ABB RAPID module: RotationTopDownTraj.MOD

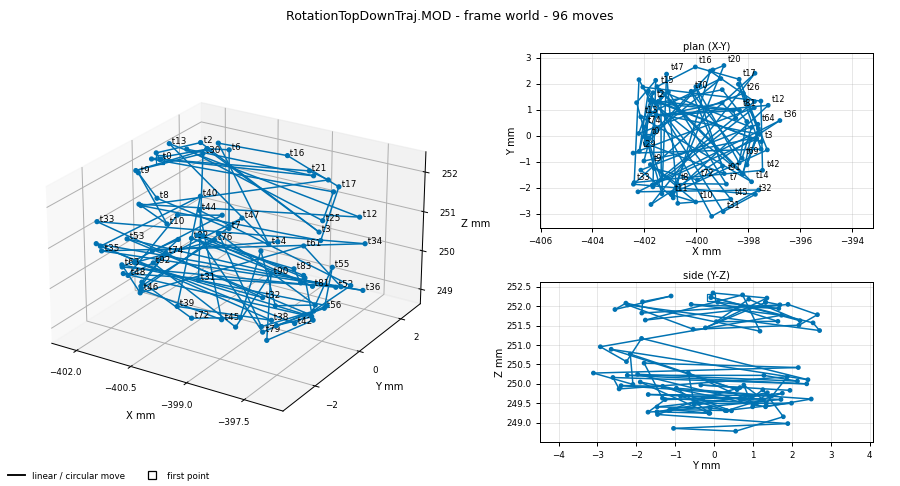
[picture p0: tool path of RotationTopDownTraj.MOD in frame world, 96 of 97 moves have a stored position in this frame; points joined in program order, loops and branches not executed]
MODULE MainModule
PERS tooldata Servo:=[TRUE,[[0,0,114.2],[1,0,0,0]],[0.215,[8.7,12.3,49.2],[1,0,0,0],0.00021,0.00024,0.00009]];
PERS tooldata tObject:=[TRUE,[[0,0,130],[0.707106781,-0.707106781,0,0]],[0.215,[8.7,12.3,49.2],[1,0,0,0],0.00021,0.00024,0.00009]];
PERS wobjdata handpos:= [FALSE,TRUE,"",[[-400,0,250],[1,0,0,0]],[[0,0,0],[1,0,0,0]]];
    PROC main()
        ConfL\Off;
        SingArea\Wrist;
        !Startpos
        MoveAbsJ [[0.441359,-16.418,10.8814,2.79121,60.2034,-14.3875],[168.362,9E+09,9E+09,9E+09,9E+09,9E+09]] \NoEOffs, v1000, fine, wi_tGripper;
        path;
    ENDPROC
    PROC path()

VAR robtarget t0 := [[-1.8594772767669543, -0.08634270627151014, 2.220359244544771], [1,0,0,0], [0,0,-1,4], [-96,9E+09,9E+09,9E+09,9E+09,9E+09]];
VAR robtarget t1 := [[-1.9968136850268585, -0.031200990620815494, 2.337895466549644], [1,0,0,0], [0,0,-1,4], [-96,9E+09,9E+09,9E+09,9E+09,9E+09]];
VAR robtarget t2 := [[-1.664406335824331, 1.3530457056262837, 2.2071876558339123], [1,0,0,0], [0,0,-1,4], [-96,9E+09,9E+09,9E+09,9E+09,9E+09]];
VAR robtarget t3 := [[2.5103465951354025, -0.22605266531133467, 1.4426248167740197], [1,0,0,0], [0,0,-1,4], [-96,9E+09,9E+09,9E+09,9E+09,9E+09]];
VAR robtarget t4 := [[-1.4698118716392545, 1.3182294867649416, 2.0926888140146214], [1,0,0,0], [0,0,-1,4], [-96,9E+09,9E+09,9E+09,9E+09,9E+09]];
VAR robtarget t5 := [[-1.4558740515764113, 1.316986954334625, 2.106495340552807], [1,0,0,0], [0,0,-1,4], [-96,9E+09,9E+09,9E+09,9E+09,9E+09]];
VAR robtarget t6 := [[-1.0750677254328767, 1.687805937624978, 2.033368826106924], [1,0,0,0], [0,0,-1,4], [-96,9E+09,9E+09,9E+09,9E+09,9E+09]];
VAR robtarget t7 := [[1.1584643511839996, -1.860619126747291, 1.8215288250970674], [1,0,0,0], [0,0,-1,4], [-96,9E+09,9E+09,9E+09,9E+09,9E+09]];
VAR robtarget t8 := [[-0.7602163155200519, -1.8412191017858337, 2.1115963079865545], [1,0,0,0], [0,0,-1,4], [-96,9E+09,9E+09,9E+09,9E+09,9E+09]];
VAR robtarget t9 := [[-1.767026063291215, -1.108222633044502, 2.2588988392369096], [1,0,0,0], [0,0,-1,4], [-96,9E+09,9E+09,9E+09,9E+09,9E+09]];
VAR robtarget t10 := [[-0.021667862335108423, -2.550518737223798, 1.91242402643374], [1,0,0,0], [0,0,-1,4], [-96,9E+09,9E+09,9E+09,9E+09,9E+09]];
VAR robtarget t11 := [[-0.9577512947057534, -2.269361244202862, 2.075411818055441], [1,0,0,0], [0,0,-1,4], [-96,9E+09,9E+09,9E+09,9E+09,9E+09]];
VAR robtarget t12 := [[2.769781059373928, 1.1748233186231039, 1.355829415691719], [1,0,0,0], [0,0,-1,4], [-96,9E+09,9E+09,9E+09,9E+09,9E+09]];
VAR robtarget t13 := [[-2.139028394244537, 0.7292214301304468, 2.2879263104279], [1,0,0,0], [0,0,-1,4], [-96,9E+09,9E+09,9E+09,9E+09,9E+09]];
VAR robtarget t14 := [[2.1287073060742876, -1.7703456012939633, 1.6407871642460183], [1,0,0,0], [0,0,-1,4], [-96,9E+09,9E+09,9E+09,9E+09,9E+09]];
VAR robtarget t15 := [[-1.513174804260462, 1.8955196047121665, 2.0442006001312616], [1,0,0,0], [0,0,-1,4], [-96,9E+09,9E+09,9E+09,9E+09,9E+09]];
VAR robtarget t16 := [[-0.03680877924259918, 2.6515244667226368, 1.7794670852935306], [1,0,0,0], [0,0,-1,4], [-96,9E+09,9E+09,9E+09,9E+09,9E+09]];
VAR robtarget t17 := [[1.6507116212087651, 2.1766451428121156, 1.5087291037843746], [1,0,0,0], [0,0,-1,4], [-96,9E+09,9E+09,9E+09,9E+09,9E+09]];
VAR robtarget t18 := [[2.735569481461933, -0.5419181356070709, 1.40601519419272], [1,0,0,0], [0,0,-1,4], [-96,9E+09,9E+09,9E+09,9E+09,9E+09]];
VAR robtarget t19 := [[-0.9380260342751103, -2.219623851546317, 2.029077273537317], [1,0,0,0], [0,0,-1,4], [-96,9E+09,9E+09,9E+09,9E+09,9E+09]];
VAR robtarget t20 := [[1.0643405616793875, 2.7065514744939527, 1.3718604556537926], [1,0,0,0], [0,0,-1,4], [-96,9E+09,9E+09,9E+09,9E+09,9E+09]];
VAR robtarget t21 := [[0.6390066698048532, 2.5391954277440463, 1.5687647182886193], [1,0,0,0], [0,0,-1,4], [-96,9E+09,9E+09,9E+09,9E+09,9E+09]];
VAR robtarget t22 := [[-1.8474595325347547, -0.0769827159651687, 2.225891768617379], [1,0,0,0], [0,0,-1,4], [-96,9E+09,9E+09,9E+09,9E+09,9E+09]];
VAR robtarget t23 := [[0.9480233018981318, 2.2051691359949985, 1.6252779556548258], [1,0,0,0], [0,0,-1,4], [-96,9E+09,9E+09,9E+09,9E+09,9E+09]];
VAR robtarget t24 := [[-1.7519363441106846, 0.8872878448625607, 2.1765162636907256], [1,0,0,0], [0,0,-1,4], [-96,9E+09,9E+09,9E+09,9E+09,9E+09]];
VAR robtarget t25 := [[2.439463854161823, 0.05449093458225296, 1.6002323474520679], [1,0,0,0], [0,0,-1,4], [-96,9E+09,9E+09,9E+09,9E+09,9E+09]];
VAR robtarget t26 := [[1.8136195796860872, 1.635838943826832, 1.607891379273222], [1,0,0,0], [0,0,-1,4], [-96,9E+09,9E+09,9E+09,9E+09,9E+09]];
VAR robtarget t27 := [[-2.2149600251011003, 0.08885764516211592, 2.0983820237528406], [1,0,0,0], [0,0,-1,4], [-96,9E+09,9E+09,9E+09,9E+09,9E+09]];
VAR robtarget t28 := [[-1.6647581164676086, 1.6588251844201465, 1.9391881751505124], [1,0,0,0], [0,0,-1,4], [-96,9E+09,9E+09,9E+09,9E+09,9E+09]];
VAR robtarget t29 := [[-2.193883206699887, -0.5920186146936126, 2.045136248873557], [1,0,0,0], [0,0,-1,4], [-96,9E+09,9E+09,9E+09,9E+09,9E+09]];
VAR robtarget t30 := [[-1.8440210325275146, 1.7282298619249423, 1.765292687731212], [1,0,0,0], [0,0,-1,4], [-96,9E+09,9E+09,9E+09,9E+09,9E+09]];
VAR robtarget t31 := [[1.0367743431461414, -2.9251234524180023, 0.9554339207288088], [1,0,0,0], [0,0,-1,4], [-96,9E+09,9E+09,9E+09,9E+09,9E+09]];
VAR robtarget t32 := [[2.275539330712497, -2.2548471355852913, 0.5737644765636434], [1,0,0,0], [0,0,-1,4], [-96,9E+09,9E+09,9E+09,9E+09,9E+09]];
VAR robtarget t33 := [[-2.420036702106024, -1.8660722061375306, 1.1696762548297064], [1,0,0,0], [0,0,-1,4], [-96,9E+09,9E+09,9E+09,9E+09,9E+09]];
VAR robtarget t34 := [[2.2605301036280805, 2.4073827316431675, 0.10883149650556624], [1,0,0,0], [0,0,-1,4], [-96,9E+09,9E+09,9E+09,9E+09,9E+09]];
VAR robtarget t35 := [[-1.7455863646872203, -2.646938022419758, 0.8908013651311293], [1,0,0,0], [0,0,-1,4], [-96,9E+09,9E+09,9E+09,9E+09,9E+09]];
VAR robtarget t36 := [[3.2195450401361567, 0.588044117864047, -0.14641264295477951], [1,0,0,0], [0,0,-1,4], [-96,9E+09,9E+09,9E+09,9E+09,9E+09]];
VAR robtarget t37 := [[-2.247320505028209, -2.15737117118444, 0.7672888712216321], [1,0,0,0], [0,0,-1,4], [-96,9E+09,9E+09,9E+09,9E+09,9E+09]];
VAR robtarget t38 := [[2.402682872066437, -2.0880962495514925, -0.01221890137512001], [1,0,0,0], [0,0,-1,4], [-96,9E+09,9E+09,9E+09,9E+09,9E+09]];
VAR robtarget t39 := [[0.5913781135054283, -3.103314944668893, 0.27937722022414974], [1,0,0,0], [0,0,-1,4], [-96,9E+09,9E+09,9E+09,9E+09,9E+09]];
VAR robtarget t40 := [[-2.207412723449383, 2.160544851459439, 0.42145624612327354], [1,0,0,0], [0,0,-1,4], [-96,9E+09,9E+09,9E+09,9E+09,9E+09]];
VAR robtarget t41 := [[-2.391079208566035, -1.8008897976182636, 0.5352609138323623], [1,0,0,0], [0,0,-1,4], [-96,9E+09,9E+09,9E+09,9E+09,9E+09]];
VAR robtarget t42 := [[2.5519092680268423, -1.3289437098540646, -0.36714326247162915], [1,0,0,0], [0,0,-1,4], [-96,9E+09,9E+09,9E+09,9E+09,9E+09]];
VAR robtarget t43 := [[2.488858861424452, 1.3374396883576571, -0.5016089742426966], [1,0,0,0], [0,0,-1,4], [-96,9E+09,9E+09,9E+09,9E+09,9E+09]];
VAR robtarget t44 := [[-2.058567611176994, 1.8766264603188998, 0.18365977136474623], [1,0,0,0], [0,0,-1,4], [-96,9E+09,9E+09,9E+09,9E+09,9E+09]];
VAR robtarget t45 := [[1.328755378691676, -2.4429884593513527, -0.12772705831947778], [1,0,0,0], [0,0,-1,4], [-96,9E+09,9E+09,9E+09,9E+09,9E+09]];
VAR robtarget t46 := [[-0.7129280245448862, -2.602204532238939, 0.16626232110087322], [1,0,0,0], [0,0,-1,4], [-96,9E+09,9E+09,9E+09,9E+09,9E+09]];
VAR robtarget t47 := [[-1.1449235497594896, 2.376210327191068, 0.00269831339624374], [1,0,0,0], [0,0,-1,4], [-96,9E+09,9E+09,9E+09,9E+09,9E+09]];
VAR robtarget t48 := [[-1.3255160472618033, -2.2327191244359508, 0.22145255025924585], [1,0,0,0], [0,0,-1,4], [-96,9E+09,9E+09,9E+09,9E+09,9E+09]];
VAR robtarget t49 := [[-2.2987884355082735, 1.2761704609581366, 0.22030620945408164], [1,0,0,0], [0,0,-1,4], [-96,9E+09,9E+09,9E+09,9E+09,9E+09]];
VAR robtarget t50 := [[-1.5642336108910437, 2.137219544705466, 0.07160528470537611], [1,0,0,0], [0,0,-1,4], [-96,9E+09,9E+09,9E+09,9E+09,9E+09]];
VAR robtarget t51 := [[-1.6699979588329499, -1.9673126444936182, 0.24788061743337053], [1,0,0,0], [0,0,-1,4], [-96,9E+09,9E+09,9E+09,9E+09,9E+09]];
VAR robtarget t52 := [[2.2347465760355116, 1.0820977650198347, -0.5064920291096195], [1,0,0,0], [0,0,-1,4], [-96,9E+09,9E+09,9E+09,9E+09,9E+09]];
VAR robtarget t53 := [[-2.4334118101716076, -0.6658255196396298, 0.2856261048295498], [1,0,0,0], [0,0,-1,4], [-96,9E+09,9E+09,9E+09,9E+09,9E+09]];
VAR robtarget t54 := [[2.496284515992172, -0.516891111642478, -0.5023960091328121], [1,0,0,0], [0,0,-1,4], [-96,9E+09,9E+09,9E+09,9E+09,9E+09]];
VAR robtarget t55 := [[1.6229339158572518, 1.9850723607230458, -0.4936291404409491], [1,0,0,0], [0,0,-1,4], [-96,9E+09,9E+09,9E+09,9E+09,9E+09]];
VAR robtarget t56 := [[2.39141814513624, 0.2812902174323957, -0.683115154681718], [1,0,0,0], [0,0,-1,4], [-96,9E+09,9E+09,9E+09,9E+09,9E+09]];
VAR robtarget t57 := [[1.9539073428531595, -1.1207916013814447, -0.656893598424261], [1,0,0,0], [0,0,-1,4], [-96,9E+09,9E+09,9E+09,9E+09,9E+09]];
VAR robtarget t58 := [[2.3010522083458262, -0.13760892674464487, -0.7519798743043697], [1,0,0,0], [0,0,-1,4], [-96,9E+09,9E+09,9E+09,9E+09,9E+09]];
VAR robtarget t59 := [[-1.6916004789630557, -1.900697654892609, 0.04984326076930095], [1,0,0,0], [0,0,-1,4], [-96,9E+09,9E+09,9E+09,9E+09,9E+09]];
VAR robtarget t60 := [[2.2401016839803085, 1.3190467116272049, -0.5860777702347993], [1,0,0,0], [0,0,-1,4], [-96,9E+09,9E+09,9E+09,9E+09,9E+09]];
VAR robtarget t61 := [[0.5353187713161721, 2.4923575287823234, -0.38744920599513466], [1,0,0,0], [0,0,-1,4], [-96,9E+09,9E+09,9E+09,9E+09,9E+09]];
VAR robtarget t62 := [[-0.8887288876717541, -2.392065552571869, -0.04382156749702511], [1,0,0,0], [0,0,-1,4], [-96,9E+09,9E+09,9E+09,9E+09,9E+09]];
VAR robtarget t63 := [[-2.1354755269462613, -1.3231065585518071, -0.05949125602243917], [1,0,0,0], [0,0,-1,4], [-96,9E+09,9E+09,9E+09,9E+09,9E+09]];
VAR robtarget t64 := [[2.3726216856142828, 0.4444016328257083, -0.6896526822853098], [1,0,0,0], [0,0,-1,4], [-96,9E+09,9E+09,9E+09,9E+09,9E+09]];
VAR robtarget t65 := [[2.327628301342003, -0.10254468018261143, -0.6164541941554126], [1,0,0,0], [0,0,-1,4], [-96,9E+09,9E+09,9E+09,9E+09,9E+09]];
VAR robtarget t66 := [[1.7651500269333018, -1.465450036977328, -0.5897479031200907], [1,0,0,0], [0,0,-1,4], [-96,9E+09,9E+09,9E+09,9E+09,9E+09]];
VAR robtarget t67 := [[-1.4298619299102704, 1.7499446809973298, -0.23831508078966362], [1,0,0,0], [0,0,-1,4], [-96,9E+09,9E+09,9E+09,9E+09,9E+09]];
VAR robtarget t68 := [[2.125499346638736, 0.3224828570183985, -0.6858150194256465], [1,0,0,0], [0,0,-1,4], [-96,9E+09,9E+09,9E+09,9E+09,9E+09]];
VAR robtarget t69 := [[1.7657607463124672, -0.8633623650517027, -0.3149630294881137], [1,0,0,0], [0,0,-1,4], [-96,9E+09,9E+09,9E+09,9E+09,9E+09]];
VAR robtarget t70 := [[-0.19657285296556215, 1.7143735903958879, -0.39850469989705156], [1,0,0,0], [0,0,-1,4], [-96,9E+09,9E+09,9E+09,9E+09,9E+09]];
VAR robtarget t71 := [[1.0138912570914276, -1.1625184255482077, -0.6836623283870141], [1,0,0,0], [0,0,-1,4], [-96,9E+09,9E+09,9E+09,9E+09,9E+09]];
VAR robtarget t72 := [[0.04313884910030008, -1.7006511619014988, -0.7249547008956304], [1,0,0,0], [0,0,-1,4], [-96,9E+09,9E+09,9E+09,9E+09,9E+09]];
VAR robtarget t73 := [[-1.6208587602714288, -1.2598497566641766, -0.40213786624185827], [1,0,0,0], [0,0,-1,4], [-96,9E+09,9E+09,9E+09,9E+09,9E+09]];
VAR robtarget t74 := [[-2.0209998343146185, 0.33763515705142044, -0.358984056927079], [1,0,0,0], [0,0,-1,4], [-96,9E+09,9E+09,9E+09,9E+09,9E+09]];
VAR robtarget t75 := [[-1.3498449650366968, -1.6948429287236437, -0.2711234372157715], [1,0,0,0], [0,0,-1,4], [-96,9E+09,9E+09,9E+09,9E+09,9E+09]];
VAR robtarget t76 := [[-1.3631235761874052, 1.4834403895031025, -0.30187647737569956], [1,0,0,0], [0,0,-1,4], [-96,9E+09,9E+09,9E+09,9E+09,9E+09]];
VAR robtarget t77 := [[-2.0169816799298275, -0.9712074610773885, -0.1093495288699723], [1,0,0,0], [0,0,-1,4], [-96,9E+09,9E+09,9E+09,9E+09,9E+09]];
VAR robtarget t78 := [[2.0907221625996506, -0.11350754806205166, -0.7536815645280284], [1,0,0,0], [0,0,-1,4], [-96,9E+09,9E+09,9E+09,9E+09,9E+09]];
VAR robtarget t79 := [[1.8020008607037572, -1.4707920119011848, -0.7164240378272466], [1,0,0,0], [0,0,-1,4], [-96,9E+09,9E+09,9E+09,9E+09,9E+09]];
VAR robtarget t80 := [[-1.7924753218201837, 1.3646862270984892, -0.22527372143072477], [1,0,0,0], [0,0,-1,4], [-96,9E+09,9E+09,9E+09,9E+09,9E+09]];
VAR robtarget t81 := [[1.6625549410710685, 0.9872631598168954, -0.5867484054084806], [1,0,0,0], [0,0,-1,4], [-96,9E+09,9E+09,9E+09,9E+09,9E+09]];
VAR robtarget t82 := [[-1.560244410944835, 0.7603313265640574, -0.02943669088350301], [1,0,0,0], [0,0,-1,4], [-96,9E+09,9E+09,9E+09,9E+09,9E+09]];
VAR robtarget t83 := [[0.9929053943143958, 1.265900992036182, -0.4079193088584916], [1,0,0,0], [0,0,-1,4], [-96,9E+09,9E+09,9E+09,9E+09,9E+09]];
VAR robtarget t84 := [[1.5210395541549393, 0.6782507543938099, -0.41275681587265634], [1,0,0,0], [0,0,-1,4], [-96,9E+09,9E+09,9E+09,9E+09,9E+09]];
VAR robtarget t85 := [[1.427602406673635, 0.9732341902123733, -0.3589070585817594], [1,0,0,0], [0,0,-1,4], [-96,9E+09,9E+09,9E+09,9E+09,9E+09]];
VAR robtarget t86 := [[-1.5612056100627998, 1.2492335701050294, -0.1465643966859974], [1,0,0,0], [0,0,-1,4], [-96,9E+09,9E+09,9E+09,9E+09,9E+09]];
VAR robtarget t87 := [[0.9989322581520983, 1.7754043089270903, -0.8423639634365613], [1,0,0,0], [0,0,-1,4], [-96,9E+09,9E+09,9E+09,9E+09,9E+09]];
VAR robtarget t88 := [[1.94437239912599, 0.5505727568418837, -1.2138160537889005], [1,0,0,0], [0,0,-1,4], [-96,9E+09,9E+09,9E+09,9E+09,9E+09]];
VAR robtarget t89 := [[1.6533463456611983, -1.0448269067267526, -1.1415065522800356], [1,0,0,0], [0,0,-1,4], [-96,9E+09,9E+09,9E+09,9E+09,9E+09]];
VAR robtarget t90 := [[-0.016648638698150364, 1.8903849060422706, -1.0182862884748802], [1,0,0,0], [0,0,-1,4], [-96,9E+09,9E+09,9E+09,9E+09,9E+09]];
VAR robtarget t91 := [[1.0753619986529983, -1.4567928725236348, -0.7844626375222101], [1,0,0,0], [0,0,-1,4], [-96,9E+09,9E+09,9E+09,9E+09,9E+09]];
VAR robtarget t92 := [[-1.9601221499167756, -0.2864223862972308, -0.36699128740678705], [1,0,0,0], [0,0,-1,4], [-96,9E+09,9E+09,9E+09,9E+09,9E+09]];
VAR robtarget t93 := [[-1.8729425710615049, 0.6605495463068062, -0.09397571869700543], [1,0,0,0], [0,0,-1,4], [-96,9E+09,9E+09,9E+09,9E+09,9E+09]];
VAR robtarget t94 := [[-1.9386388127720695, -0.34376279223466844, -0.02749651531651455], [1,0,0,0], [0,0,-1,4], [-96,9E+09,9E+09,9E+09,9E+09,9E+09]];
VAR robtarget t95 := [[0.1354703220075713, 1.9456575161450018, -0.16454634957136155], [1,0,0,0], [0,0,-1,4], [-96,9E+09,9E+09,9E+09,9E+09,9E+09]];MoveL t0, v100\V:=100.000, z1, wi_tGripper, \WObj:=handpos;
MoveL t1, v100\V:=100.000, z1, wi_tGripper, \WObj:=handpos;
MoveL t2, v100\V:=100.000, z1, wi_tGripper, \WObj:=handpos;
MoveL t3, v100\V:=100.000, z1, wi_tGripper, \WObj:=handpos;
MoveL t4, v100\V:=100.000, z1, wi_tGripper, \WObj:=handpos;
MoveL t5, v100\V:=100.000, z1, wi_tGripper, \WObj:=handpos;
MoveL t6, v100\V:=100.000, z1, wi_tGripper, \WObj:=handpos;
MoveL t7, v100\V:=100.000, z1, wi_tGripper, \WObj:=handpos;
MoveL t8, v100\V:=100.000, z1, wi_tGripper, \WObj:=handpos;
MoveL t9, v100\V:=100.000, z1, wi_tGripper, \WObj:=handpos;
MoveL t10, v100\V:=100.000, z1, wi_tGripper, \WObj:=handpos;
MoveL t11, v100\V:=100.000, z1, wi_tGripper, \WObj:=handpos;
MoveL t12, v100\V:=100.000, z1, wi_tGripper, \WObj:=handpos;
MoveL t13, v100\V:=100.000, z1, wi_tGripper, \WObj:=handpos;
MoveL t14, v100\V:=100.000, z1, wi_tGripper, \WObj:=handpos;
MoveL t15, v100\V:=100.000, z1, wi_tGripper, \WObj:=handpos;
MoveL t16, v100\V:=100.000, z1, wi_tGripper, \WObj:=handpos;
MoveL t17, v100\V:=100.000, z1, wi_tGripper, \WObj:=handpos;
MoveL t18, v100\V:=100.000, z1, wi_tGripper, \WObj:=handpos;
MoveL t19, v100\V:=100.000, z1, wi_tGripper, \WObj:=handpos;
MoveL t20, v100\V:=100.000, z1, wi_tGripper, \WObj:=handpos;
MoveL t21, v100\V:=100.000, z1, wi_tGripper, \WObj:=handpos;
MoveL t22, v100\V:=100.000, z1, wi_tGripper, \WObj:=handpos;
MoveL t23, v100\V:=100.000, z1, wi_tGripper, \WObj:=handpos;
MoveL t24, v100\V:=100.000, z1, wi_tGripper, \WObj:=handpos;
MoveL t25, v100\V:=100.000, z1, wi_tGripper, \WObj:=handpos;
MoveL t26, v100\V:=100.000, z1, wi_tGripper, \WObj:=handpos;
MoveL t27, v100\V:=100.000, z1, wi_tGripper, \WObj:=handpos;
MoveL t28, v100\V:=100.000, z1, wi_tGripper, \WObj:=handpos;
MoveL t29, v100\V:=100.000, z1, wi_tGripper, \WObj:=handpos;
MoveL t30, v100\V:=100.000, z1, wi_tGripper, \WObj:=handpos;
MoveL t31, v100\V:=100.000, z1, wi_tGripper, \WObj:=handpos;
MoveL t32, v100\V:=100.000, z1, wi_tGripper, \WObj:=handpos;
MoveL t33, v100\V:=100.000, z1, wi_tGripper, \WObj:=handpos;
MoveL t34, v100\V:=100.000, z1, wi_tGripper, \WObj:=handpos;
MoveL t35, v100\V:=100.000, z1, wi_tGripper, \WObj:=handpos;
MoveL t36, v100\V:=100.000, z1, wi_tGripper, \WObj:=handpos;
MoveL t37, v100\V:=100.000, z1, wi_tGripper, \WObj:=handpos;
MoveL t38, v100\V:=100.000, z1, wi_tGripper, \WObj:=handpos;
MoveL t39, v100\V:=100.000, z1, wi_tGripper, \WObj:=handpos;
MoveL t40, v100\V:=100.000, z1, wi_tGripper, \WObj:=handpos;
MoveL t41, v100\V:=100.000, z1, wi_tGripper, \WObj:=handpos;
MoveL t42, v100\V:=100.000, z1, wi_tGripper, \WObj:=handpos;
MoveL t43, v100\V:=100.000, z1, wi_tGripper, \WObj:=handpos;
MoveL t44, v100\V:=100.000, z1, wi_tGripper, \WObj:=handpos;
MoveL t45, v100\V:=100.000, z1, wi_tGripper, \WObj:=handpos;
MoveL t46, v100\V:=100.000, z1, wi_tGripper, \WObj:=handpos;
MoveL t47, v100\V:=100.000, z1, wi_tGripper, \WObj:=handpos;
MoveL t48, v100\V:=100.000, z1, wi_tGripper, \WObj:=handpos;
MoveL t49, v100\V:=100.000, z1, wi_tGripper, \WObj:=handpos;
MoveL t50, v100\V:=100.000, z1, wi_tGripper, \WObj:=handpos;
MoveL t51, v100\V:=100.000, z1, wi_tGripper, \WObj:=handpos;
MoveL t52, v100\V:=100.000, z1, wi_tGripper, \WObj:=handpos;
MoveL t53, v100\V:=100.000, z1, wi_tGripper, \WObj:=handpos;
MoveL t54, v100\V:=100.000, z1, wi_tGripper, \WObj:=handpos;
MoveL t55, v100\V:=100.000, z1, wi_tGripper, \WObj:=handpos;
MoveL t56, v100\V:=100.000, z1, wi_tGripper, \WObj:=handpos;
MoveL t57, v100\V:=100.000, z1, wi_tGripper, \WObj:=handpos;
MoveL t58, v100\V:=100.000, z1, wi_tGripper, \WObj:=handpos;
MoveL t59, v100\V:=100.000, z1, wi_tGripper, \WObj:=handpos;
MoveL t60, v100\V:=100.000, z1, wi_tGripper, \WObj:=handpos;
MoveL t61, v100\V:=100.000, z1, wi_tGripper, \WObj:=handpos;
MoveL t62, v100\V:=100.000, z1, wi_tGripper, \WObj:=handpos;
MoveL t63, v100\V:=100.000, z1, wi_tGripper, \WObj:=handpos;
MoveL t64, v100\V:=100.000, z1, wi_tGripper, \WObj:=handpos;
MoveL t65, v100\V:=100.000, z1, wi_tGripper, \WObj:=handpos;
MoveL t66, v100\V:=100.000, z1, wi_tGripper, \WObj:=handpos;
MoveL t67, v100\V:=100.000, z1, wi_tGripper, \WObj:=handpos;
MoveL t68, v100\V:=100.000, z1, wi_tGripper, \WObj:=handpos;
MoveL t69, v100\V:=100.000, z1, wi_tGripper, \WObj:=handpos;
MoveL t70, v100\V:=100.000, z1, wi_tGripper, \WObj:=handpos;
MoveL t71, v100\V:=100.000, z1, wi_tGripper, \WObj:=handpos;
MoveL t72, v100\V:=100.000, z1, wi_tGripper, \WObj:=handpos;
MoveL t73, v100\V:=100.000, z1, wi_tGripper, \WObj:=handpos;
MoveL t74, v100\V:=100.000, z1, wi_tGripper, \WObj:=handpos;
MoveL t75, v100\V:=100.000, z1, wi_tGripper, \WObj:=handpos;
MoveL t76, v100\V:=100.000, z1, wi_tGripper, \WObj:=handpos;
MoveL t77, v100\V:=100.000, z1, wi_tGripper, \WObj:=handpos;
MoveL t78, v100\V:=100.000, z1, wi_tGripper, \WObj:=handpos;
MoveL t79, v100\V:=100.000, z1, wi_tGripper, \WObj:=handpos;
MoveL t80, v100\V:=100.000, z1, wi_tGripper, \WObj:=handpos;
MoveL t81, v100\V:=100.000, z1, wi_tGripper, \WObj:=handpos;
MoveL t82, v100\V:=100.000, z1, wi_tGripper, \WObj:=handpos;
MoveL t83, v100\V:=100.000, z1, wi_tGripper, \WObj:=handpos;
MoveL t84, v100\V:=100.000, z1, wi_tGripper, \WObj:=handpos;
MoveL t85, v100\V:=100.000, z1, wi_tGripper, \WObj:=handpos;
MoveL t86, v100\V:=100.000, z1, wi_tGripper, \WObj:=handpos;
MoveL t87, v100\V:=100.000, z1, wi_tGripper, \WObj:=handpos;
MoveL t88, v100\V:=100.000, z1, wi_tGripper, \WObj:=handpos;
MoveL t89, v100\V:=100.000, z1, wi_tGripper, \WObj:=handpos;
MoveL t90, v100\V:=100.000, z1, wi_tGripper, \WObj:=handpos;
MoveL t91, v100\V:=100.000, z1, wi_tGripper, \WObj:=handpos;
MoveL t92, v100\V:=100.000, z1, wi_tGripper, \WObj:=handpos;
MoveL t93, v100\V:=100.000, z1, wi_tGripper, \WObj:=handpos;
MoveL t94, v100\V:=100.000, z1, wi_tGripper, \WObj:=handpos;
MoveL t95, v100\V:=100.000, z1, wi_tGripper, \WObj:=handpos;

ENDPROC
ENDMODULE
